// ---- POUs/DALI/DALI_Setup/VISUs/Visu_DALICommissioning/Visu_Part102Groups.TcVIS
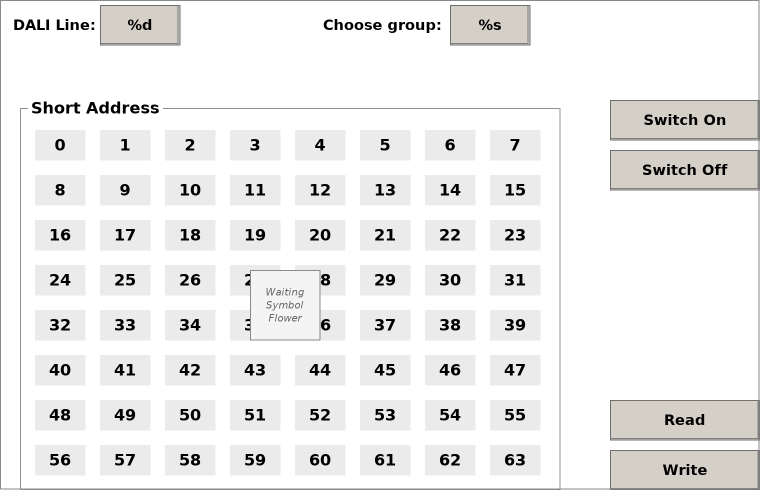
VISUALIZATION Visu_Part102Groups  // 760x490
    GroupBox (20,100 540x390), "Short Address"
        Textfield (15,30 50x30), "0", colour toggle: DALI_Commissioning.fbPart102Groups.aShowAlarmState[0] = TRUE, invisible if: DALI_Commissioning.fbPart102Groups.aActivateButton[0] = FALSE, input disabled if: DALI_Commissioning.fbPart102Groups.aActivateButton[0] = FALSE
            OnMouseClick: execute { DALI_Commissioning.fbPart102Groups.aButtonClick[0] := TRUE; }
        Textfield (80,30 50x30), "1", colour toggle: DALI_Commissioning.fbPart102Groups.aShowAlarmState[1] = TRUE, invisible if: DALI_Commissioning.fbPart102Groups.aActivateButton[1] = FALSE, input disabled if: DALI_Commissioning.fbPart102Groups.aActivateButton[1] = FALSE
            OnMouseClick: execute { DALI_Commissioning.fbPart102Groups.aButtonClick[1] := TRUE; }
        Textfield (145,30 50x30), "2", colour toggle: DALI_Commissioning.fbPart102Groups.aShowAlarmState[2] = TRUE, invisible if: DALI_Commissioning.fbPart102Groups.aActivateButton[2] = FALSE, input disabled if: DALI_Commissioning.fbPart102Groups.aActivateButton[2] = FALSE
            OnMouseClick: execute { DALI_Commissioning.fbPart102Groups.aButtonClick[2] := TRUE; }
        Textfield (210,30 50x30), "3", colour toggle: DALI_Commissioning.fbPart102Groups.aShowAlarmState[3] = TRUE, invisible if: DALI_Commissioning.fbPart102Groups.aActivateButton[3] = FALSE, input disabled if: DALI_Commissioning.fbPart102Groups.aActivateButton[3] = FALSE
            OnMouseClick: execute { DALI_Commissioning.fbPart102Groups.aButtonClick[3] := TRUE; }
        Textfield (275,30 50x30), "4", colour toggle: DALI_Commissioning.fbPart102Groups.aShowAlarmState[4] = TRUE, invisible if: DALI_Commissioning.fbPart102Groups.aActivateButton[4] = FALSE, input disabled if: DALI_Commissioning.fbPart102Groups.aActivateButton[4] = FALSE
            OnMouseClick: execute { DALI_Commissioning.fbPart102Groups.aButtonClick[4] := TRUE; }
        Textfield (340,30 50x30), "5", colour toggle: DALI_Commissioning.fbPart102Groups.aShowAlarmState[5] = TRUE, invisible if: DALI_Commissioning.fbPart102Groups.aActivateButton[5] = FALSE, input disabled if: DALI_Commissioning.fbPart102Groups.aActivateButton[5] = FALSE
            OnMouseClick: execute { DALI_Commissioning.fbPart102Groups.aButtonClick[5] := TRUE; }
        Textfield (405,30 50x30), "6", colour toggle: DALI_Commissioning.fbPart102Groups.aShowAlarmState[6] = TRUE, invisible if: DALI_Commissioning.fbPart102Groups.aActivateButton[6] = FALSE, input disabled if: DALI_Commissioning.fbPart102Groups.aActivateButton[6] = FALSE
            OnMouseClick: execute { DALI_Commissioning.fbPart102Groups.aButtonClick[6] := TRUE; }
        Textfield (470,30 50x30), "7", colour toggle: DALI_Commissioning.fbPart102Groups.aShowAlarmState[7] = TRUE, invisible if: DALI_Commissioning.fbPart102Groups.aActivateButton[7] = FALSE, input disabled if: DALI_Commissioning.fbPart102Groups.aActivateButton[7] = FALSE
            OnMouseClick: execute { DALI_Commissioning.fbPart102Groups.aButtonClick[7] := TRUE; }
        Textfield (15,75 50x30), "8", colour toggle: DALI_Commissioning.fbPart102Groups.aShowAlarmState[8] = TRUE, invisible if: DALI_Commissioning.fbPart102Groups.aActivateButton[8] = FALSE, input disabled if: DALI_Commissioning.fbPart102Groups.aActivateButton[8] = FALSE
            OnMouseClick: execute { DALI_Commissioning.fbPart102Groups.aButtonClick[8] := TRUE; }
        Textfield (80,75 50x30), "9", colour toggle: DALI_Commissioning.fbPart102Groups.aShowAlarmState[9] = TRUE, invisible if: DALI_Commissioning.fbPart102Groups.aActivateButton[9] = FALSE, input disabled if: DALI_Commissioning.fbPart102Groups.aActivateButton[9] = FALSE
            OnMouseClick: execute { DALI_Commissioning.fbPart102Groups.aButtonClick[9] := TRUE; }
        Textfield (145,75 50x30), "10", colour toggle: DALI_Commissioning.fbPart102Groups.aShowAlarmState[10] = TRUE, invisible if: DALI_Commissioning.fbPart102Groups.aActivateButton[10] = FALSE, input disabled if: DALI_Commissioning.fbPart102Groups.aActivateButton[10] = FALSE
            OnMouseClick: execute { DALI_Commissioning.fbPart102Groups.aButtonClick[10] := TRUE; }
        Textfield (210,75 50x30), "11", colour toggle: DALI_Commissioning.fbPart102Groups.aShowAlarmState[11] = TRUE, invisible if: DALI_Commissioning.fbPart102Groups.aActivateButton[11] = FALSE, input disabled if: DALI_Commissioning.fbPart102Groups.aActivateButton[11] = FALSE
            OnMouseClick: execute { DALI_Commissioning.fbPart102Groups.aButtonClick[11] := TRUE; }
        Textfield (275,75 50x30), "12", colour toggle: DALI_Commissioning.fbPart102Groups.aShowAlarmState[12] = TRUE, invisible if: DALI_Commissioning.fbPart102Groups.aActivateButton[12] = FALSE, input disabled if: DALI_Commissioning.fbPart102Groups.aActivateButton[12] = FALSE
            OnMouseClick: execute { DALI_Commissioning.fbPart102Groups.aButtonClick[12] := TRUE; }
        Textfield (340,75 50x30), "13", colour toggle: DALI_Commissioning.fbPart102Groups.aShowAlarmState[13] = TRUE, invisible if: DALI_Commissioning.fbPart102Groups.aActivateButton[13] = FALSE, input disabled if: DALI_Commissioning.fbPart102Groups.aActivateButton[13] = FALSE
            OnMouseClick: execute { DALI_Commissioning.fbPart102Groups.aButtonClick[13] := TRUE; }
        Textfield (405,75 50x30), "14", colour toggle: DALI_Commissioning.fbPart102Groups.aShowAlarmState[14] = TRUE, invisible if: DALI_Commissioning.fbPart102Groups.aActivateButton[14] = FALSE, input disabled if: DALI_Commissioning.fbPart102Groups.aActivateButton[14] = FALSE
            OnMouseClick: execute { DALI_Commissioning.fbPart102Groups.aButtonClick[14] := TRUE; }
        Textfield (470,75 50x30), "15", colour toggle: DALI_Commissioning.fbPart102Groups.aShowAlarmState[15] = TRUE, invisible if: DALI_Commissioning.fbPart102Groups.aActivateButton[15] = FALSE, input disabled if: DALI_Commissioning.fbPart102Groups.aActivateButton[15] = FALSE
            OnMouseClick: execute { DALI_Commissioning.fbPart102Groups.aButtonClick[15] := TRUE; }
        Textfield (15,120 50x30), "16", colour toggle: DALI_Commissioning.fbPart102Groups.aShowAlarmState[16] = TRUE, invisible if: DALI_Commissioning.fbPart102Groups.aActivateButton[16] = FALSE, input disabled if: DALI_Commissioning.fbPart102Groups.aActivateButton[16] = FALSE
            OnMouseClick: execute { DALI_Commissioning.fbPart102Groups.aButtonClick[16] := TRUE; }
        Textfield (80,120 50x30), "17", colour toggle: DALI_Commissioning.fbPart102Groups.aShowAlarmState[17] = TRUE, invisible if: DALI_Commissioning.fbPart102Groups.aActivateButton[17] = FALSE, input disabled if: DALI_Commissioning.fbPart102Groups.aActivateButton[17] = FALSE
            OnMouseClick: execute { DALI_Commissioning.fbPart102Groups.aButtonClick[17] := TRUE; }
        Textfield (145,120 50x30), "18", colour toggle: DALI_Commissioning.fbPart102Groups.aShowAlarmState[18] = TRUE, invisible if: DALI_Commissioning.fbPart102Groups.aActivateButton[18] = FALSE, input disabled if: DALI_Commissioning.fbPart102Groups.aActivateButton[18] = FALSE
            OnMouseClick: execute { DALI_Commissioning.fbPart102Groups.aButtonClick[18] := TRUE; }
        Textfield (210,120 50x30), "19", colour toggle: DALI_Commissioning.fbPart102Groups.aShowAlarmState[19] = TRUE, invisible if: DALI_Commissioning.fbPart102Groups.aActivateButton[19] = FALSE, input disabled if: DALI_Commissioning.fbPart102Groups.aActivateButton[19] = FALSE
            OnMouseClick: execute { DALI_Commissioning.fbPart102Groups.aButtonClick[19] := TRUE; }
        Textfield (275,120 50x30), "20", colour toggle: DALI_Commissioning.fbPart102Groups.aShowAlarmState[20] = TRUE, invisible if: DALI_Commissioning.fbPart102Groups.aActivateButton[20] = FALSE, input disabled if: DALI_Commissioning.fbPart102Groups.aActivateButton[20] = FALSE
            OnMouseClick: execute { DALI_Commissioning.fbPart102Groups.aButtonClick[20] := TRUE; }
        Textfield (340,120 50x30), "21", colour toggle: DALI_Commissioning.fbPart102Groups.aShowAlarmState[21] = TRUE, invisible if: DALI_Commissioning.fbPart102Groups.aActivateButton[21] = FALSE, input disabled if: DALI_Commissioning.fbPart102Groups.aActivateButton[21] = FALSE
            OnMouseClick: execute { DALI_Commissioning.fbPart102Groups.aButtonClick[21] := TRUE; }
        Textfield (405,120 50x30), "22", colour toggle: DALI_Commissioning.fbPart102Groups.aShowAlarmState[22] = TRUE, invisible if: DALI_Commissioning.fbPart102Groups.aActivateButton[22] = FALSE, input disabled if: DALI_Commissioning.fbPart102Groups.aActivateButton[22] = FALSE
            OnMouseClick: execute { DALI_Commissioning.fbPart102Groups.aButtonClick[22] := TRUE; }
        Textfield (470,120 50x30), "23", colour toggle: DALI_Commissioning.fbPart102Groups.aShowAlarmState[23] = TRUE, invisible if: DALI_Commissioning.fbPart102Groups.aActivateButton[23] = FALSE, input disabled if: DALI_Commissioning.fbPart102Groups.aActivateButton[23] = FALSE
            OnMouseClick: execute { DALI_Commissioning.fbPart102Groups.aButtonClick[23] := TRUE; }
        Textfield (15,165 50x30), "24", colour toggle: DALI_Commissioning.fbPart102Groups.aShowAlarmState[24] = TRUE, invisible if: DALI_Commissioning.fbPart102Groups.aDeviceGroupState[24] = 0, input disabled if: DALI_Commissioning.fbPart102Groups.aDeviceGroupState[24] = 0
            OnMouseClick: execute { DALI_Commissioning.fbPart102Groups.aButtonClick[24] := TRUE; }
        Textfield (80,165 50x30), "25", colour toggle: DALI_Commissioning.fbPart102Groups.aShowAlarmState[25] = TRUE, invisible if: DALI_Commissioning.fbPart102Groups.aActivateButton[25] = FALSE, input disabled if: DALI_Commissioning.fbPart102Groups.aActivateButton[25] = FALSE
            OnMouseClick: execute { DALI_Commissioning.fbPart102Groups.aButtonClick[25] := TRUE; }
        Textfield (145,165 50x30), "26", colour toggle: DALI_Commissioning.fbPart102Groups.aShowAlarmState[26] = TRUE, invisible if: DALI_Commissioning.fbPart102Groups.aActivateButton[26] = FALSE, input disabled if: DALI_Commissioning.fbPart102Groups.aActivateButton[26] = FALSE
            OnMouseClick: execute { DALI_Commissioning.fbPart102Groups.aButtonClick[26] := TRUE; }
        Textfield (210,165 50x30), "27", colour toggle: DALI_Commissioning.fbPart102Groups.aShowAlarmState[27] = TRUE, invisible if: DALI_Commissioning.fbPart102Groups.aActivateButton[27] = FALSE, input disabled if: DALI_Commissioning.fbPart102Groups.aActivateButton[27] = FALSE
            OnMouseClick: execute { DALI_Commissioning.fbPart102Groups.aButtonClick[27] := TRUE; }
        Textfield (275,165 50x30), "28", colour toggle: DALI_Commissioning.fbPart102Groups.aShowAlarmState[28] = TRUE, invisible if: DALI_Commissioning.fbPart102Groups.aActivateButton[28] = FALSE, input disabled if: DALI_Commissioning.fbPart102Groups.aActivateButton[28] = FALSE
            OnMouseClick: execute { DALI_Commissioning.fbPart102Groups.aButtonClick[28] := TRUE; }
        Textfield (340,165 50x30), "29", colour toggle: DALI_Commissioning.fbPart102Groups.aShowAlarmState[29] = TRUE, invisible if: DALI_Commissioning.fbPart102Groups.aActivateButton[29] = FALSE, input disabled if: DALI_Commissioning.fbPart102Groups.aActivateButton[29] = FALSE
            OnMouseClick: execute { DALI_Commissioning.fbPart102Groups.aButtonClick[29] := TRUE; }
        Textfield (405,165 50x30), "30", colour toggle: DALI_Commissioning.fbPart102Groups.aShowAlarmState[30] = TRUE, invisible if: DALI_Commissioning.fbPart102Groups.aActivateButton[30] = FALSE, input disabled if: DALI_Commissioning.fbPart102Groups.aActivateButton[30] = FALSE
            OnMouseClick: execute { DALI_Commissioning.fbPart102Groups.aButtonClick[30] := TRUE; }
        Textfield (470,165 50x30), "31", colour toggle: DALI_Commissioning.fbPart102Groups.aShowAlarmState[31] = TRUE, invisible if: DALI_Commissioning.fbPart102Groups.aActivateButton[31] = FALSE, input disabled if: DALI_Commissioning.fbPart102Groups.aActivateButton[31] = FALSE
            OnMouseClick: execute { DALI_Commissioning.fbPart102Groups.aButtonClick[31] := TRUE; }
        Textfield (15,210 50x30), "32", colour toggle: DALI_Commissioning.fbPart102Groups.aShowAlarmState[32] = TRUE, invisible if: DALI_Commissioning.fbPart102Groups.aActivateButton[32] = FALSE, input disabled if: DALI_Commissioning.fbPart102Groups.aActivateButton[32] = FALSE
            OnMouseClick: execute { DALI_Commissioning.fbPart102Groups.aButtonClick[32] := TRUE; }
        Textfield (80,210 50x30), "33", colour toggle: DALI_Commissioning.fbPart102Groups.aShowAlarmState[33] = TRUE, invisible if: DALI_Commissioning.fbPart102Groups.aActivateButton[33] = FALSE, input disabled if: DALI_Commissioning.fbPart102Groups.aActivateButton[33] = FALSE
            OnMouseClick: execute { DALI_Commissioning.fbPart102Groups.aButtonClick[33] := TRUE; }
        Textfield (145,210 50x30), "34", colour toggle: DALI_Commissioning.fbPart102Groups.aShowAlarmState[34] = TRUE, invisible if: DALI_Commissioning.fbPart102Groups.aActivateButton[34] = FALSE, input disabled if: DALI_Commissioning.fbPart102Groups.aActivateButton[34] = FALSE
            OnMouseClick: execute { DALI_Commissioning.fbPart102Groups.aButtonClick[34] := TRUE; }
        Textfield (210,210 50x30), "35", colour toggle: DALI_Commissioning.fbPart102Groups.aShowAlarmState[35] = TRUE, invisible if: DALI_Commissioning.fbPart102Groups.aActivateButton[35] = FALSE, input disabled if: DALI_Commissioning.fbPart102Groups.aActivateButton[35] = FALSE
            OnMouseClick: execute { DALI_Commissioning.fbPart102Groups.aButtonClick[35] := TRUE; }
        Textfield (275,210 50x30), "36", colour toggle: DALI_Commissioning.fbPart102Groups.aShowAlarmState[36] = TRUE, invisible if: DALI_Commissioning.fbPart102Groups.aActivateButton[36] = FALSE, input disabled if: DALI_Commissioning.fbPart102Groups.aActivateButton[36] = FALSE
            OnMouseClick: execute { DALI_Commissioning.fbPart102Groups.aButtonClick[36] := TRUE; }
        Textfield (340,210 50x30), "37", colour toggle: DALI_Commissioning.fbPart102Groups.aShowAlarmState[37] = TRUE, invisible if: DALI_Commissioning.fbPart102Groups.aActivateButton[37] = FALSE, input disabled if: DALI_Commissioning.fbPart102Groups.aActivateButton[37] = FALSE
            OnMouseClick: execute { DALI_Commissioning.fbPart102Groups.aButtonClick[37] := TRUE; }
        Textfield (405,210 50x30), "38", colour toggle: DALI_Commissioning.fbPart102Groups.aShowAlarmState[38] = TRUE, invisible if: DALI_Commissioning.fbPart102Groups.aActivateButton[38] = FALSE, input disabled if: DALI_Commissioning.fbPart102Groups.aActivateButton[38] = FALSE
            OnMouseClick: execute { DALI_Commissioning.fbPart102Groups.aButtonClick[38] := TRUE; }
        Textfield (470,210 50x30), "39", colour toggle: DALI_Commissioning.fbPart102Groups.aShowAlarmState[39] = TRUE, invisible if: DALI_Commissioning.fbPart102Groups.aActivateButton[39] = FALSE, input disabled if: DALI_Commissioning.fbPart102Groups.aActivateButton[39] = FALSE
            OnMouseClick: execute { DALI_Commissioning.fbPart102Groups.aButtonClick[39] := TRUE; }
        Textfield (15,255 50x30), "40", colour toggle: DALI_Commissioning.fbPart102Groups.aShowAlarmState[40] = TRUE, invisible if: DALI_Commissioning.fbPart102Groups.aActivateButton[40] = FALSE, input disabled if: DALI_Commissioning.fbPart102Groups.aActivateButton[40] = FALSE
            OnMouseClick: execute { DALI_Commissioning.fbPart102Groups.aButtonClick[40] := TRUE; }
        Textfield (80,255 50x30), "41", colour toggle: DALI_Commissioning.fbPart102Groups.aShowAlarmState[41] = TRUE, invisible if: DALI_Commissioning.fbPart102Groups.aActivateButton[41] = FALSE, input disabled if: DALI_Commissioning.fbPart102Groups.aActivateButton[41] = FALSE
            OnMouseClick: execute { DALI_Commissioning.fbPart102Groups.aButtonClick[41] := TRUE; }
        Textfield (145,255 50x30), "42", colour toggle: DALI_Commissioning.fbPart102Groups.aShowAlarmState[42] = TRUE, invisible if: DALI_Commissioning.fbPart102Groups.aActivateButton[42] = FALSE, input disabled if: DALI_Commissioning.fbPart102Groups.aActivateButton[42] = FALSE
            OnMouseClick: execute { DALI_Commissioning.fbPart102Groups.aButtonClick[42] := TRUE; }
        Textfield (210,255 50x30), "43", colour toggle: DALI_Commissioning.fbPart102Groups.aShowAlarmState[43] = TRUE, invisible if: DALI_Commissioning.fbPart102Groups.aActivateButton[43] = FALSE, input disabled if: DALI_Commissioning.fbPart102Groups.aActivateButton[43] = FALSE
            OnMouseClick: execute { DALI_Commissioning.fbPart102Groups.aButtonClick[43] := TRUE; }
        Textfield (275,255 50x30), "44", colour toggle: DALI_Commissioning.fbPart102Groups.aShowAlarmState[44] = TRUE, invisible if: DALI_Commissioning.fbPart102Groups.aActivateButton[44] = FALSE, input disabled if: DALI_Commissioning.fbPart102Groups.aActivateButton[44] = FALSE
            OnMouseClick: execute { DALI_Commissioning.fbPart102Groups.aButtonClick[44] := TRUE; }
        Textfield (340,255 50x30), "45", colour toggle: DALI_Commissioning.fbPart102Groups.aShowAlarmState[45] = TRUE, invisible if: DALI_Commissioning.fbPart102Groups.aActivateButton[45] = FALSE, input disabled if: DALI_Commissioning.fbPart102Groups.aActivateButton[45] = FALSE
            OnMouseClick: execute { DALI_Commissioning.fbPart102Groups.aButtonClick[45] := TRUE; }
        Textfield (405,255 50x30), "46", colour toggle: DALI_Commissioning.fbPart102Groups.aShowAlarmState[46] = TRUE, invisible if: DALI_Commissioning.fbPart102Groups.aActivateButton[46] = FALSE, input disabled if: DALI_Commissioning.fbPart102Groups.aActivateButton[46] = FALSE
            OnMouseClick: execute { DALI_Commissioning.fbPart102Groups.aButtonClick[46] := TRUE; }
        Textfield (470,255 50x30), "47", colour toggle: DALI_Commissioning.fbPart102Groups.aShowAlarmState[47] = TRUE, invisible if: DALI_Commissioning.fbPart102Groups.aActivateButton[47] = FALSE, input disabled if: DALI_Commissioning.fbPart102Groups.aActivateButton[47] = FALSE
            OnMouseClick: execute { DALI_Commissioning.fbPart102Groups.aButtonClick[47] := TRUE; }
        Textfield (15,300 50x30), "48", colour toggle: DALI_Commissioning.fbPart102Groups.aShowAlarmState[48] = TRUE, invisible if: DALI_Commissioning.fbPart102Groups.aActivateButton[48] = FALSE, input disabled if: DALI_Commissioning.fbPart102Groups.aActivateButton[48] = FALSE
            OnMouseClick: execute { DALI_Commissioning.fbPart102Groups.aButtonClick[48] := TRUE; }
        Textfield (80,300 50x30), "49", colour toggle: DALI_Commissioning.fbPart102Groups.aShowAlarmState[49] = TRUE, invisible if: DALI_Commissioning.fbPart102Groups.aActivateButton[49] = FALSE, input disabled if: DALI_Commissioning.fbPart102Groups.aActivateButton[49] = FALSE
            OnMouseClick: execute { DALI_Commissioning.fbPart102Groups.aButtonClick[49] := TRUE; }
        Textfield (145,300 50x30), "50", colour toggle: DALI_Commissioning.fbPart102Groups.aShowAlarmState[50] = TRUE, invisible if: DALI_Commissioning.fbPart102Groups.aActivateButton[50] = FALSE, input disabled if: DALI_Commissioning.fbPart102Groups.aActivateButton[50] = FALSE
            OnMouseClick: execute { DALI_Commissioning.fbPart102Groups.aButtonClick[50] := TRUE; }
        Textfield (210,300 50x30), "51", colour toggle: DALI_Commissioning.fbPart102Groups.aShowAlarmState[51] = TRUE, invisible if: DALI_Commissioning.fbPart102Groups.aActivateButton[51] = FALSE, input disabled if: DALI_Commissioning.fbPart102Groups.aActivateButton[51] = FALSE
            OnMouseClick: execute { DALI_Commissioning.fbPart102Groups.aButtonClick[51] := TRUE; }
        Textfield (275,300 50x30), "52", colour toggle: DALI_Commissioning.fbPart102Groups.aShowAlarmState[52] = TRUE, invisible if: DALI_Commissioning.fbPart102Groups.aActivateButton[52] = FALSE, input disabled if: DALI_Commissioning.fbPart102Groups.aActivateButton[52] = FALSE
            OnMouseClick: execute { DALI_Commissioning.fbPart102Groups.aButtonClick[52] := TRUE; }
        Textfield (340,300 50x30), "53", colour toggle: DALI_Commissioning.fbPart102Groups.aShowAlarmState[53] = TRUE, invisible if: DALI_Commissioning.fbPart102Groups.aActivateButton[53] = FALSE, input disabled if: DALI_Commissioning.fbPart102Groups.aActivateButton[53] = FALSE
            OnMouseClick: execute { DALI_Commissioning.fbPart102Groups.aButtonClick[53] := TRUE; }
        Textfield (405,300 50x30), "54", colour toggle: DALI_Commissioning.fbPart102Groups.aShowAlarmState[54] = TRUE, invisible if: DALI_Commissioning.fbPart102Groups.aActivateButton[54] = FALSE, input disabled if: DALI_Commissioning.fbPart102Groups.aActivateButton[54] = FALSE
            OnMouseClick: execute { DALI_Commissioning.fbPart102Groups.aButtonClick[54] := TRUE; }
        Textfield (470,300 50x30), "55", colour toggle: DALI_Commissioning.fbPart102Groups.aShowAlarmState[55] = TRUE, invisible if: DALI_Commissioning.fbPart102Groups.aActivateButton[55] = FALSE, input disabled if: DALI_Commissioning.fbPart102Groups.aActivateButton[55] = FALSE
            OnMouseClick: execute { DALI_Commissioning.fbPart102Groups.aButtonClick[55] := TRUE; }
        Textfield (15,345 50x30), "56", colour toggle: DALI_Commissioning.fbPart102Groups.aShowAlarmState[56] = TRUE, invisible if: DALI_Commissioning.fbPart102Groups.aActivateButton[56] = FALSE, input disabled if: DALI_Commissioning.fbPart102Groups.aActivateButton[56] = FALSE
            OnMouseClick: execute { DALI_Commissioning.fbPart102Groups.aButtonClick[56] := TRUE; }
        Textfield (80,345 50x30), "57", colour toggle: DALI_Commissioning.fbPart102Groups.aShowAlarmState[57] = TRUE, invisible if: DALI_Commissioning.fbPart102Groups.aActivateButton[57] = FALSE, input disabled if: DALI_Commissioning.fbPart102Groups.aActivateButton[57] = FALSE
            OnMouseClick: execute { DALI_Commissioning.fbPart102Groups.aButtonClick[56] := TRUE; }
        Textfield (145,345 50x30), "58", colour toggle: DALI_Commissioning.fbPart102Groups.aShowAlarmState[58] = TRUE, invisible if: DALI_Commissioning.fbPart102Groups.aActivateButton[58] = FALSE, input disabled if: DALI_Commissioning.fbPart102Groups.aActivateButton[58] = FALSE
            OnMouseClick: execute { DALI_Commissioning.fbPart102Groups.aButtonClick[58] := TRUE; }
        Textfield (210,345 50x30), "59", colour toggle: DALI_Commissioning.fbPart102Groups.aShowAlarmState[59] = TRUE, invisible if: DALI_Commissioning.fbPart102Groups.aActivateButton[59] = FALSE, input disabled if: DALI_Commissioning.fbPart102Groups.aActivateButton[59] = FALSE
            OnMouseClick: execute { DALI_Commissioning.fbPart102Groups.aButtonClick[59] := TRUE; }
        Textfield (275,345 50x30), "60", colour toggle: DALI_Commissioning.fbPart102Groups.aShowAlarmState[60] = TRUE, invisible if: DALI_Commissioning.fbPart102Groups.aActivateButton[60] = FALSE, input disabled if: DALI_Commissioning.fbPart102Groups.aActivateButton[60] = FALSE
            OnMouseClick: execute { DALI_Commissioning.fbPart102Groups.aButtonClick[60] := TRUE; }
        Textfield (340,345 50x30), "61", colour toggle: DALI_Commissioning.fbPart102Groups.aShowAlarmState[61] = TRUE, invisible if: DALI_Commissioning.fbPart102Groups.aActivateButton[61] = FALSE, input disabled if: DALI_Commissioning.fbPart102Groups.aActivateButton[61] = FALSE
            OnMouseClick: execute { DALI_Commissioning.fbPart102Groups.aButtonClick[61] := TRUE; }
        Textfield (405,345 50x30), "62", colour toggle: DALI_Commissioning.fbPart102Groups.aShowAlarmState[62] = TRUE, invisible if: DALI_Commissioning.fbPart102Groups.aActivateButton[62] = FALSE, input disabled if: DALI_Commissioning.fbPart102Groups.aActivateButton[62] = FALSE
            OnMouseClick: execute { DALI_Commissioning.fbPart102Groups.aButtonClick[62] := TRUE; }
        Textfield (470,345 50x30), "63", colour toggle: DALI_Commissioning.fbPart102Groups.aShowAlarmState[63] = TRUE, invisible if: DALI_Commissioning.fbPart102Groups.aActivateButton[63] = FALSE, input disabled if: DALI_Commissioning.fbPart102Groups.aActivateButton[63] = FALSE
            OnMouseClick: execute { DALI_Commissioning.fbPart102Groups.aButtonClick[63] := TRUE; }
        WaitingSymbolFlower (230,170 70x70), invisible if: DALI_Commissioning.fbPart102Groups.bHideWaitSymbol
    Button (610,400 150x40), "Read"
        OnMouseClick: execute { DALI_Commissioning.fbPart102Groups.bRead := TRUE; }
    Button (610,450 150x40), "Write"
        OnMouseClick: execute { DALI_Commissioning.fbPart102Groups.bWrite := TRUE; }
    Button (610,100 150x40), "Switch On"
        OnMouseClick: execute { DALI_Commissioning.fbPart102Groups.bSwitchOn := TRUE; }
    Button (610,150 150x40), "Switch Off"
        OnMouseClick: execute { DALI_Commissioning.fbPart102Groups.bSwitchOff := TRUE; }
    Group (320,5 210x40)
        Textfield (0,0 120x40), "Choose group:"
        Button (130,0 80x40), "%s", text variable: DALI_Commissioning.fbPart102Groups.nGroupAddress
            OnMouseClick: write the text variable via Default, min 0, max 15, title "Choose group"
    Group (10,5 170x40)
        Textfield (0,0 110x40), "DALI Line:"
        Button (90,0 80x40), "%d", text variable: GVL_Internal.nDALILine
            OnMouseClick: write the text variable via Default, min 1, max 10, title "Choose line"
END_VISUALIZATION

// ---- POUs/DALI/DALI_Setup/VISUs/Visu_DALICommissioning/Visu_Part103Addressing.TcVIS
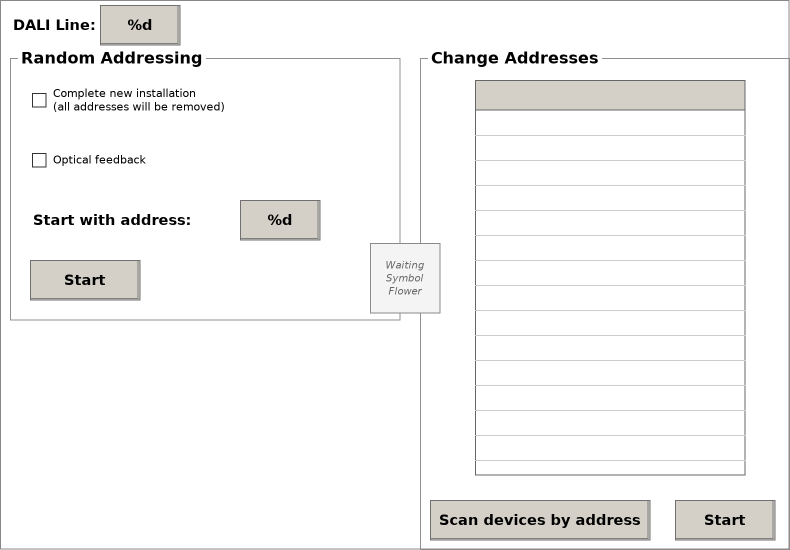
VISUALIZATION Visu_Part103Addressing  // 790x550
    GroupBox (420,50 370x500), "Change Addresses"
        Table (55,30 270x395), data array: DALI_Commissioning.fbPart103Addressing.aChangeAddressList
            p3854506369: DALI_Commissioning.fbPart103Addressing.aChangeAddressList[INDEX].nOldAddress
            p1892666644: DALI_Commissioning.fbPart103Addressing.aChangeAddressList[INDEX].nNewAddress
            p338671338: DALI_Commissioning.fbPart103Addressing.aChangeAddressList[INDEX].nRandomAddress
            p2170511999: DALI_Commissioning.fbPart103Addressing.aChangeAddressList[INDEX].nErrors
            Columns.Column.[0].Template: DALI_Commissioning.fbPart103Addressing.aNoShortAddress[INDEX]
            Columns.Column.[1].Template: DALI_Commissioning.fbPart103Addressing.aNoShortAddress[INDEX]; OnMouseClick: write the text variable via Default, min 0, max 63, title "New Short Address"
        Button (255,450 100x40), "Start"
            OnMouseClick: execute { DALI_Commissioning.fbPart103Addressing.bStartChangeAddress := TRUE; }
        Button (10,450 220x40), "Scan devices by address"
            OnMouseClick: execute { DALI_Commissioning.fbPart103Addressing.bScanDevices := TRUE; }
    GroupBox (10,50 390x270), "Random Addressing"
        Button (20,210 110x40), "Start"
            OnMouseClick: execute { DALI_Commissioning.fbPart103Addressing.bStartRandomAddressing := TRUE; }
        Checkbox (20,30 360x40), "Complete new installation (all addresses will be removed)", variable: DALI_Commissioning.fbPart103Addressing.bNewInstallation
        Checkbox (20,90 360x40), "Optical feedback", variable: DALI_Commissioning.fbPart103Addressing.bOpticalFeedback
        Textfield (20,150 200x40), "Start with address:"
        Button (230,150 80x40), "%d", text variable: DALI_Commissioning.fbPart103Addressing.nStartAddress
            OnMouseClick: write DALI_Commissioning.fbPart103Addressing.nStartAddress via Default, min 0, max 63, title "Insert Short Address"
    WaitingSymbolFlower (370,243 70x70), invisible if: DALI_Commissioning.fbPart103Addressing.bHideWaitSymbol
    Group (10,5 170x40)
        Textfield (0,0 110x40), "DALI Line:"
        Button (90,0 80x40), "%d", text variable: GVL_Internal.nDALILine
            OnMouseClick: write the text variable via Default, min 1, max 10, title "Choose line"
END_VISUALIZATION

// ---- POUs/DALI/DALI_Setup/VISUs/Visu_DALICommissioning/Visu_Part103Identify.TcVIS
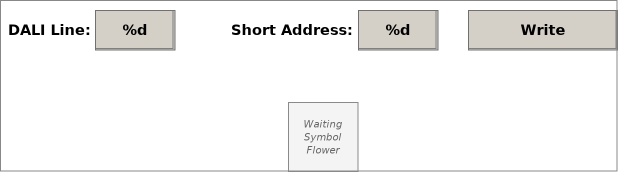
VISUALIZATION Visu_Part103Identify  // 618x172
    Button (468,10 150x40), "Write"
        OnMouseClick: execute { DALI_Commissioning.fbPart103IdentifyDevice.bWrite := TRUE; }
    WaitingSymbolFlower (288,102 70x70), invisible if: DALI_Commissioning.fbPart103MemoryPages.bHideWaitSymbol
    Textfield (228,10 130x40), "Short Address:"
    Button (358,10 80x40), "%d", text variable: DALI_Commissioning.fbPart103IdentifyDevice.nAddress
        OnMouseClick: write the text variable via Default, min 0, max 63, title "Insert Short Address"
    Group (5,10 170x40)
        Textfield (0,0 110x40), "DALI Line:"
        Button (90,0 80x40), "%d", text variable: GVL_Internal.nDALILine
            OnMouseClick: write the text variable via Default, min 1, max 10, title "Choose line"
END_VISUALIZATION

// ---- POUs/DALI/DALI_Setup/VISUs/Visu_DALICommissioning/Visu_Part202.TcVIS
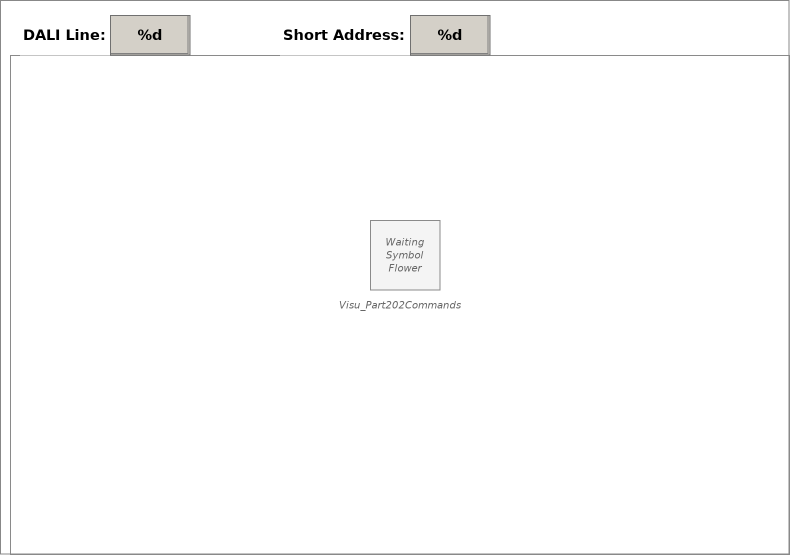
VISUALIZATION Visu_Part202  // 790x555
    TabControl (10,55 780x500)
        shows Visu_Part202Commands()
        shows Visu_Part202Status()
        shows Visu_Part202Parameters()
        [0]: TabTitle=Commands
        [1]: TabTitle=Status
        [2]: TabTitle=Parameters
    Group (280,15 210x40)
        Textfield (0,0 130x40), "Short Address:"
        Button (130,0 80x40), "%d", text variable: DALI_Commissioning.fbPart202Emergency.nAddress
            OnMouseClick: write the text variable via Default, min 0, max 63, title "Insert Short Address"
    Group (20,15 170x40)
        Textfield (0,0 110x40), "DALI Line:"
        Button (90,0 80x40), "%d", text variable: GVL_Internal.nDALILine
            OnMouseClick: write the text variable via Default, min 1, max 10, title "Choose line"
    WaitingSymbolFlower (370,220 70x70), invisible if: DALI_Commissioning.fbPart202Emergency.bHideWaitSymbol
END_VISUALIZATION

// ---- POUs/DALI/DALI_Setup/VISUs/Visu_DALICommissioning/Visu_Part208Switching.TcVIS
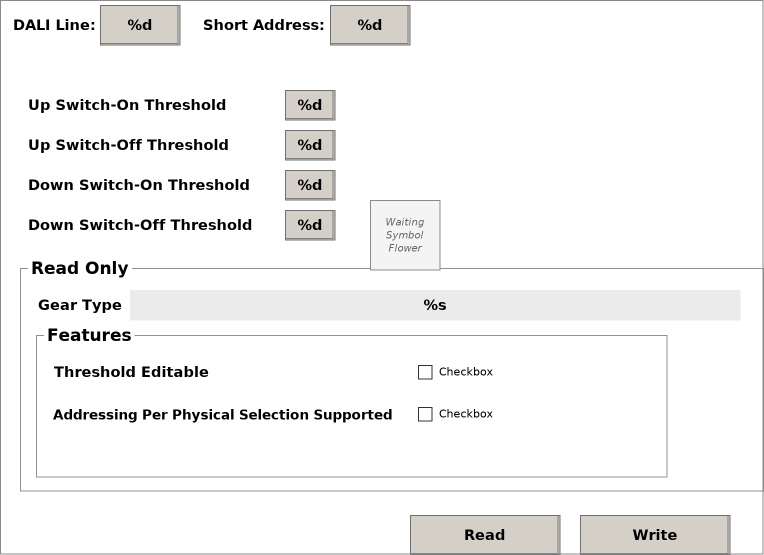
VISUALIZATION Visu_Part208Switching  // 764x555
    Group (200,5 210x40)
        Textfield (0,0 130x40), "Short Address:"
        Button (130,0 80x40), "%d", text variable: DALI_Commissioning.fbPart208Switching.nAddress
            OnMouseClick: write the text variable via Default, min 0, max 63, title "Insert Short Address"
    Group (10,5 170x40)
        Textfield (0,0 110x40), "DALI Line:"
        Button (90,0 80x40), "%d", text variable: GVL_Internal.nDALILine
            OnMouseClick: write the text variable via Default, min 1, max 10, title "Choose line"
    Textfield (25,90 250x30), "Up Switch-On Threshold"
    Textfield (25,130 250x30), "Up Switch-Off Threshold"
    Textfield (25,170 250x30), "Down Switch-On Threshold"
    Textfield (25,210 250x30), "Down Switch-Off Threshold"
    GroupBox (20,260 744x231), "Read Only"
        Textfield (15,30 250x30), "Gear Type"
        Textfield (110,30 610x30), "%s", text variable: DALI_Commissioning.fbPart208Switching.sGearType
        GroupBox (16,67 631x150), "Features"
            Checkbox (380,30 30x30), "Checkbox", variable: DALI_Commissioning.fbPart208Switching.bThreshold, input disabled if: TRUE
            Textfield (15,30 350x30), "Threshold Editable"
            Checkbox (380,72 30x30), "Checkbox", variable: DALI_Commissioning.fbPart208Switching.bAddressingPhysical, input disabled if: TRUE
    Textfield (50,400 355x30), "Addressing Per Physical Selection Supported"
    Button (410,515 150x40), "Read"
        OnMouseClick: execute { DALI_Commissioning.fbPart208Switching.bRead := TRUE; }
    Button (580,515 150x40), "Write"
        OnMouseClick: execute { DALI_Commissioning.fbPart208Switching.bWrite := TRUE; }
    WaitingSymbolFlower (370,200 70x70), invisible if: DALI_Commissioning.fbPart208Switching.bHideWaitSymbol
    Button (285,90 50x30), "%d", text variable: DALI_Commissioning.fbPart208Switching.nUpSwitchOnThreshold
        OnMouseClick: write the text variable via Default, min 0, max 255, title "Up Switch On Threshold"
    Button (285,130 50x30), "%d", text variable: DALI_Commissioning.fbPart208Switching.nUpSwitchOffThreshold
        OnMouseClick: write the text variable via Default, min 0, max 255, title "Up Switch Off Threshold"
    Button (285,170 50x30), "%d", text variable: DALI_Commissioning.fbPart208Switching.nDownSwitchOnThreshold
        OnMouseClick: write the text variable via Default, min 0, max 255, title "Down Switch On Threshold"
    Button (285,210 50x30), "%d", text variable: DALI_Commissioning.fbPart208Switching.nDownSwitchOffThreshold
        OnMouseClick: write the text variable via Default, min 0, max 255, title "Down Switch Off Threshold"
END_VISUALIZATION

// ---- POUs/DALI/DALI_Setup/VISUs/Visu_DALICommissioning/Visu_Part300GenericDevice.TcVIS
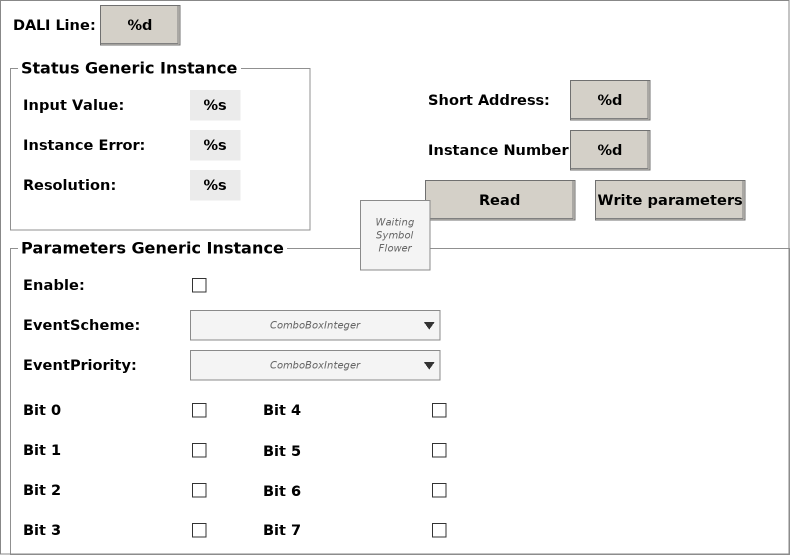
VISUALIZATION Visu_Part300GenericDevice  // 790x555
    GroupBox (10,240 780x315), "Parameters Generic Instance"
        Textfield (10,30 150x30), "Enable:"
        Checkbox (180,30 30x30), variable: DALI_Commissioning.fbPart300GenericDevice.bEnable
        Textfield (10,110 150x30), "EventPriority:"
        Textfield (10,195 100x30), "Bit 1"
        Textfield (10,155 100x30), "Bit 0"
        Checkbox (180,155 30x30), variable: DALI_Commissioning.fbPart300GenericDevice.bBit0
        Checkbox (180,195 30x30), variable: DALI_Commissioning.fbPart300GenericDevice.bBit1
        Textfield (10,235 100x30), "Bit 2"
        Textfield (250,155 100x30), "Bit 4"
        Textfield (250,196 100x30), "Bit 5"
        Checkbox (420,195 30x30), variable: DALI_Commissioning.fbPart300GenericDevice.bBit5
        Checkbox (420,155 30x30), variable: DALI_Commissioning.fbPart300GenericDevice.bBit4
        Checkbox (180,275 30x30), variable: DALI_Commissioning.fbPart300GenericDevice.bBit3
        Checkbox (180,235 30x30), variable: DALI_Commissioning.fbPart300GenericDevice.bBit2
        ComboBoxInteger (180,70 250x30), variable: DALI_Commissioning.fbPart300GenericDevice.eEventScheme, text list: 'EventScheme'
        Textfield (10,70 150x30), "EventScheme:"
        Textfield (250,236 100x30), "Bit 6"
        ComboBoxInteger (180,110 250x30), variable: DALI_Commissioning.fbPart300GenericDevice.eEventPriority, text list: 'EventPriority'
        Textfield (10,275 100x30), "Bit 3"
        Checkbox (420,235 30x30), variable: DALI_Commissioning.fbPart300GenericDevice.bBit6
        Checkbox (420,275 30x30), variable: DALI_Commissioning.fbPart300GenericDevice.bBit7
        Textfield (250,275 100x30), "Bit 7"
    GroupBox (10,60 300x170), "Status Generic Instance"
        Textfield (180,30 50x30), "%s", text variable: DALI_Commissioning.fbPart300GenericDevice.nInputValue
        Textfield (180,70 50x30), "%s", text variable: DALI_Commissioning.fbPart300GenericDevice.nInstanceError
        Textfield (180,110 50x30), "%s", text variable: DALI_Commissioning.fbPart300GenericDevice.nResolution
        Textfield (10,30 160x30), "Input Value:"
        Textfield (10,70 160x30), "Instance Error:"
        Textfield (10,110 160x30), "Resolution:"
    Button (425,180 150x40), "Read"
        OnMouseClick: execute { DALI_Commissioning.fbPart300GenericDevice.bRead := TRUE; }
    WaitingSymbolFlower (360,200 70x70), invisible if: DALI_Commissioning.fbPart300GenericDevice.bHideWaitSymbol
    Button (595,180 150x40), "Write parameters"
        OnMouseClick: execute { DALI_Commissioning.fbPart300GenericDevice.bWrite := TRUE; }
    Textfield (425,130 150x40), "Instance Number:"
    Textfield (425,80 150x40), "Short Address:"
    Button (570,80 80x40), "%d", text variable: DALI_Commissioning.fbPart300GenericDevice.nAddress
        OnMouseClick: write the text variable via Default, min 0, max 63, title "Insert Short Address"
    Button (570,130 80x40), "%d", text variable: DALI_Commissioning.fbPart300GenericDevice.nInstanceAddress
        OnMouseClick: write the text variable via Default, min 0, max 31, title "Insert instance number"
    Group (10,5 170x40)
        Textfield (0,0 110x40), "DALI Line:"
        Button (90,0 80x40), "%d", text variable: GVL_Internal.nDALILine
            OnMouseClick: write the text variable via Default, min 1, max 10, title "Choose line"
END_VISUALIZATION

// ---- POUs/DALI/DALI_Setup/VISUs/Visu_DALICommissioning/Visu_Part301PushButton.TcVIS
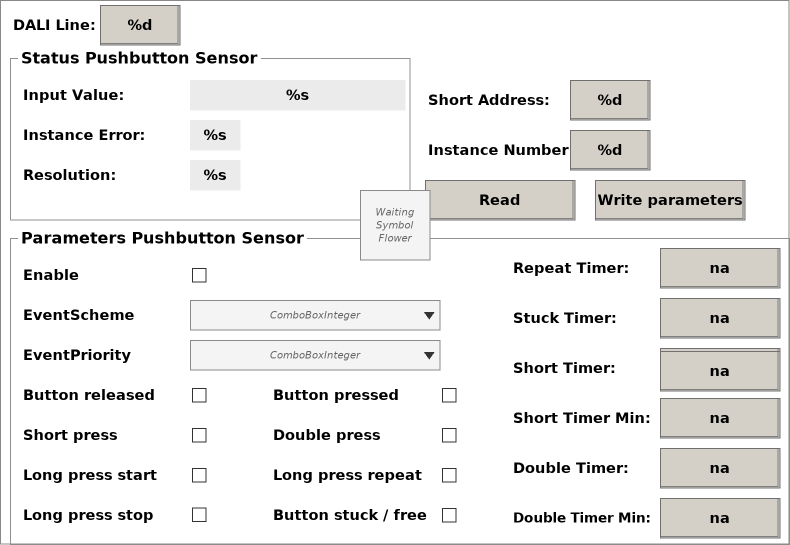
VISUALIZATION Visu_Part301PushButton  // 790x545
    GroupBox (10,230 780x315), "Parameters Pushbutton Sensor"
        Button (650,268 120x40), "%d ms", text variable: DALI_Commissioning.fbPart301PushButton.nDoubleMin
        Button (650,268 120x40), "na", invisible if: Not DALI_Commissioning.fbPart301PushButton.bNoDoubleTimer, input disabled if: Not DALI_Commissioning.fbPart301PushButton.bNoDoubleTimer
        Button (650,168 120x40), "%d ms", text variable: DALI_Commissioning.fbPart301PushButton.nShortMin
        Button (650,168 120x40), "na", invisible if: Not DALI_Commissioning.fbPart301PushButton.bNoRepeatTimer, input disabled if: Not DALI_Commissioning.fbPart301PushButton.bNoRepeatTimer
        Button (650,218 120x40), "%d ms", text variable: DALI_Commissioning.fbPart301PushButton.nDouble
            OnMouseClick: write the text variable via Default, min 0, max 2000, title "Insert value for double timer"
        Button (650,218 120x40), "na", invisible if: Not DALI_Commissioning.fbPart301PushButton.bNoDoubleTimer, input disabled if: Not DALI_Commissioning.fbPart301PushButton.bNoDoubleTimer
        Button (650,118 120x40), "%d ms", text variable: DALI_Commissioning.fbPart301PushButton.nShort
            OnMouseClick: write the text variable via Default, min 10, max 500, title "Insert value for short timer"
        Button (650,121 120x40), "na", invisible if: Not DALI_Commissioning.fbPart301PushButton.bNoRepeatTimer, input disabled if: Not DALI_Commissioning.fbPart301PushButton.bNoRepeatTimer
        Button (650,68 120x40), "%d s", text variable: DALI_Commissioning.fbPart301PushButton.nStuck
            OnMouseClick: write the text variable via Default, min 5, max 255, title "Insert value for stuck timer"
        Button (650,68 120x40), "na", invisible if: Not DALI_Commissioning.fbPart301PushButton.bNoRepeatTimer, input disabled if: Not DALI_Commissioning.fbPart301PushButton.bNoRepeatTimer
        Button (650,18 120x40), "%d ms", text variable: DALI_Commissioning.fbPart301PushButton.nRepeat
            OnMouseClick: write the text variable via Default, min 100, max 2000, title "Insert value for repeat timer"
        Button (650,18 120x40), "na", invisible if: Not DALI_Commissioning.fbPart301PushButton.bNoRepeatTimer, input disabled if: Not DALI_Commissioning.fbPart301PushButton.bNoRepeatTimer
        Textfield (500,23 145x30), "Repeat Timer:"
        Textfield (500,73 145x30), "Stuck Timer:"
        Textfield (500,123 145x30), "Short Timer:"
        Textfield (500,223 145x30), "Double Timer:"
        Textfield (10,30 170x30), "Enable"
        Checkbox (180,30 30x30), variable: DALI_Commissioning.fbPart301PushButton.bEnable
        Textfield (10,70 170x30), "EventScheme"
        Textfield (10,150 170x30), "Button released"
        Textfield (10,190 170x30), "Short press"
        Textfield (10,230 170x30), "Long press start"
        Textfield (10,270 170x30), "Long press stop"
        Textfield (260,150 170x30), "Button pressed"
        Textfield (260,190 170x30), "Double press"
        Textfield (260,230 170x30), "Long press repeat"
        Textfield (260,270 170x30), "Button stuck / free"
        Checkbox (180,150 30x30), variable: DALI_Commissioning.fbPart301PushButton.bButtonReleased
        Checkbox (180,190 30x30), variable: DALI_Commissioning.fbPart301PushButton.bShortPress
        Checkbox (180,230 30x30), variable: DALI_Commissioning.fbPart301PushButton.bLongPressStart
        Checkbox (430,150 30x30), variable: DALI_Commissioning.fbPart301PushButton.bButtonPressed
        Checkbox (430,190 30x30), variable: DALI_Commissioning.fbPart301PushButton.bDoublePress
        Checkbox (430,230 29x30), variable: DALI_Commissioning.fbPart301PushButton.bLongPressRepeat
        Checkbox (430,270 30x30), variable: DALI_Commissioning.fbPart301PushButton.bButtonStuck
        ComboBoxInteger (180,70 250x30), variable: DALI_Commissioning.fbPart301PushButton.eEventScheme, text list: 'EventScheme'
        Checkbox (180,270 28x29), variable: DALI_Commissioning.fbPart301PushButton.bLongPressStop
        Textfield (10,110 170x30), "EventPriority"
        ComboBoxInteger (180,110 250x30), variable: DALI_Commissioning.fbPart301PushButton.eEventPriority, text list: 'EventPriority'
        Textfield (500,173 145x30), "Short Timer Min:"
        Textfield (500,273 145x30), "Double Timer Min:"
    GroupBox (10,50 400x170), "Status Pushbutton Sensor"
        Textfield (10,30 160x30), "Input Value:"
        Textfield (10,70 160x30), "Instance Error:"
        Textfield (10,110 160x30), "Resolution:"
        Textfield (180,30 215x30), "%s", text variable: DALI_Commissioning.fbPart301PushButton.sInputValue
        Textfield (180,70 50x30), "%s", text variable: DALI_Commissioning.fbPart301PushButton.nInstanceError
        Textfield (180,110 50x30), "%s", text variable: DALI_Commissioning.fbPart301PushButton.nResolution
    Button (425,180 150x40), "Read"
        OnMouseClick: execute { DALI_Commissioning.fbPart301PushButton.bRead := TRUE; }
    WaitingSymbolFlower (360,190 70x70), invisible if: DALI_Commissioning.fbPart301PushButton.bHideWaitSymbol
    Button (595,180 150x40), "Write parameters"
        OnMouseClick: execute { DALI_Commissioning.fbPart301PushButton.bWrite := TRUE; }
    Group (10,5 170x40)
        Textfield (0,0 110x40), "DALI Line:"
        Button (90,0 80x40), "%d", text variable: GVL_Internal.nDALILine
            OnMouseClick: write the text variable via Default, min 1, max 10, title "Choose line"
    Textfield (425,80 160x40), "Short Address:"
    Button (570,80 80x40), "%d", text variable: DALI_Commissioning.fbPart301PushButton.nAddress
        OnMouseClick: write the text variable via Default, min 0, max 63, title "Insert Short Address"
    Textfield (425,130 150x40), "Instance Number:"
    Button (570,130 80x40), "%d", text variable: DALI_Commissioning.fbPart301PushButton.nInstanceAddress
        OnMouseClick: write the text variable via Default, min 0, max 31, title "Insert instance number"
END_VISUALIZATION
